// TIA Portal V18 export
TYPE "MEStoPLC_MainCheckInStation1ST350_Laser"
// stored: IsFailsafeCompliant false
   STRUCT
      PartTypeID : Int;   // Part type ID extracted from part type description
      Station1PalletID : Int;   // Pallet ID
      Station1PartSN : String[60];   // Serial number - Housing
      Spare : Array[0..132] of Byte;   // 备用
      Massage : "MEStoPLC_AlarmMassage_ext";   // Process error code
      LaserMarking { S7_SetPoint := 'True'} : "LaserMarkingBuffer";
   END_STRUCT;
END_TYPE
